FUNCTION_BLOCK DrillStation
  (* Standard: 61499-2 *)
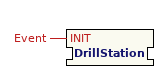
  EVENT_INPUT
    INIT;
  END_EVENT
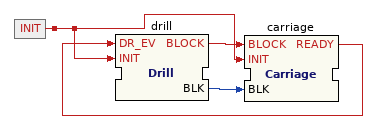
  FBS
    drill : Drill;
    carriage : Carriage;
  END_FBS
  EVENT_CONNECTIONS
    drill.BLOCK TO carriage.BLOCK;
    carriage.READY TO drill.DR_EV;
    INIT TO drill.INIT;
    INIT TO carriage.INIT;
  END_CONNECTIONS
  DATA_CONNECTIONS
    drill.BLK TO carriage.BLK;
  END_CONNECTIONS
END_FUNCTION_BLOCK
